TYPE ST_ProtectionSystems_Params :
STRUCT
	InsulationMonitor				: ST_InsulationMonitor_params;
	firedetection					: ST_Firedetection_params;
	OCP								: ST_Overcurrentprotection_params;
END_STRUCT
END_TYPE

(* stored: Version 1.1.0.1, ProductVersion 3.1.4026.18
   DUT ST_ProtectionSystems_Params: Id {b5cb0580-39d7-4160-bf35-6357b189c45e} *)
